FUNCTION_BLOCK MUL_INT (* IEC 61131-3 INT Multiplication *)
  (* Standard: 61131-3 *)
  (* Version 0.0, 2004-12-15, JHC, Rockwell Automation, Converted from SRC format. *)
  (* Compiler header: package fb.rt.plc.math; *)
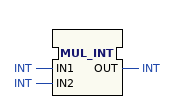
  VAR_INPUT
    IN1 : INT; (* Multiplicand *)
    IN2 : INT; (* Multiplier *)
  END_VAR
  VAR_OUTPUT
    OUT : INT; (* Product *)
  END_VAR
END_FUNCTION_BLOCK
